FUNCTION_BLOCK _REAL_TestSuite EXTENDS TcUnit.FB_TestSuite
VAR
END_VAR

TestAddress();
TestClearReference();
TestClone();
TestTypeNameReturnsExpected();
TestIsFloat();
TestIsSigned();
TestMakeReferenceToFollowsReference();
TestMakeReferenceToUpdatesReference();
TestSize();
TestValueReturnsExpectedAfterInit();
TestValueReturnsExpectedAfterChange();
TestSerializeTypeWith();
TestSerializeWith();
TestTryDeserializeFrom();
TestTryMakeReferenceToFollowsReference();
TestTryMakeReferenceToUpdatesReference();

METHOD PUBLIC TestAddress
VAR
    _type : _REAL(0.0);
    notExpected : PVOID := 0;
    actual : PVOID;
END_VAR
TEST('TestAddress');

actual := _type.Address;

AssertFalse(
    Condition := (notExpected = actual),
    Message := 'Type did not return a valid address.'
);

TEST_FINISHED();
END_METHOD

METHOD PUBLIC TestClearReference
VAR
    _type : _REAL(0.0);
	target : REAL := 0.0;
    expected : REAL := 0.0;
    actual : REAL;
END_VAR
TEST('TestClearReference');

_type.MakeReferenceTo(target);
_type.ClearReference();
target := 123.4;

actual := _type.Value;

AssertEquals_REAL(
    Expected := expected,
    Actual := actual,
    Delta := REAL#0.001,
    Message := 'Value incorrectly followed target change'
);

TEST_FINISHED();
END_METHOD

METHOD PUBLIC TestClone
VAR
    _type : _REAL(123.4);
	clone : I_Datatype;
	isValidClone : BOOL;
	compareResult : DINT;
END_VAR
TEST('TestClone');

clone := _type.Clone();

isValidClone := clone <> 0;

IF isValidClone THEN
	compareResult := memcmp(_type.Address, clone.Address, clone.Size);
END_IF

AssertTrue(
	Condition := isValidClone,
	Message := 'Clone did not produce a clone'
);

AssertEquals_DINT(
	Expected := 0,
    Actual := compareResult,
    Message := 'Clone did not return a valid clone.'
);

clone.Dispose();

TEST_FINISHED();
END_METHOD

METHOD PUBLIC TestIsFloat
VAR
    _type : _REAL(0);
END_VAR
TEST('TestIsFloat');

AssertTrue(
	Condition := _type.IsFloat,
    Message := 'Type did not correctly identify itself as being unsigned'
);

TEST_FINISHED();
END_METHOD

METHOD PUBLIC TestIsSigned
VAR
    _type : _REAL(0);
END_VAR
TEST('TestIsSigned');

AssertTrue(
	Condition := _type.IsSigned,
    Message := 'Type did not correctly identify itself as being signed'
);

TEST_FINISHED();
END_METHOD

METHOD PUBLIC TestMakeReferenceToFollowsReference
VAR
    _type : _REAL(0.0);
	target : REAL := 0.0;
    expected : REAL := 123.4;
    actual : REAL;
END_VAR
TEST('TestMakeReferenceToFollowsReference');

_type.MakeReferenceTo(target);
target := 123.4;

actual := _type.Value;

AssertEquals_REAL(
    Expected := expected,
    Actual := actual,
    Delta := REAL#0.001,
    Message := 'Value did not follow target change'
);

TEST_FINISHED();
END_METHOD

METHOD PUBLIC TestMakeReferenceToUpdatesReference
VAR
    _type : _REAL(0.0);
	target : REAL := 0.0;
    expected : REAL := 123.4;
    actual : REAL;
END_VAR
TEST('TestMakeReferenceToUpdatesReference');

_type.MakeReferenceTo(target);
_type.Value := 123.4;

actual := target;

AssertEquals_REAL(
    Expected := expected,
    Actual := actual,
    Delta := REAL#0.001,
    Message := 'Value did not update target'
);

TEST_FINISHED();
END_METHOD

METHOD PUBLIC TestSerializeTypeWith
VAR
    _type : _REAL(0.0);
    serializer : JsonSerializer;
    expected : STRING(500) := '{"typeName":"REAL","minValue":-3.4028230607370967e38,"maxValue":3.4028230607370967e38,"isSigned":true,"isFloat":true}';
    actual : STRING(500);
END_VAR
TEST('TestSerializeTypeWith');

serializer.Reset();
_type.SerializeTypeWith(serializer);
serializer.TryGetSerializedData(ADR(actual), SIZEOF(actual));

AssertEquals_STRING(
    Expected := expected,
    Actual := actual,
    Message := 'Serialization of type did not return correct string.'
);

TEST_FINISHED();
END_METHOD

METHOD PUBLIC TestSerializeWith
VAR
    _type : _REAL(123.4);
    serializer : JsonSerializer;
    expected : STRING := '123.4000015258789'; // Expected value due to the nature of floating point values defined by IEEE754.
    actual : STRING(500);
END_VAR
TEST('TestSerializeWith');

serializer.Reset();
_type.SerializeWith(serializer);
serializer.TryGetSerializedData(ADR(actual), SIZEOF(actual));

AssertEquals_STRING(
    Expected := expected,
    Actual := actual,
    Message := 'Serialization of type data did not return correct string.'
);

TEST_FINISHED();
END_METHOD

METHOD PUBLIC TestSize
VAR
    _type : _REAL(0.0);
    expected : UDINT := SIZEOF(REAL);
    actual : UDINT;
END_VAR
TEST('TestSize');

actual := _type.Size;

AssertEquals_UDINT(
    Expected := Expected,
    Actual := actual,
    Message := 'Type did not return the correct size.'
);

TEST_FINISHED();
END_METHOD

METHOD PUBLIC TestTryDeserializeFrom
VAR
    deserializer : JsonDeserializer;
    feedback : DeserializerFeedback;
    json : STRING := '123.4';
    _type : _REAL(0.0);
    expected : REAL := 123.4;
    actual : REAL;
 END_VAR
TEST('TestTryDeserializeFrom');

deserializer.Reset();
deserializer.TryLoad(json);
_type.TryDeserializeFrom(Deserializer, Feedback);

actual := _type.Value;

AssertEquals_REAL(
    Expected := expected,
    Actual := actual,
    Delta := REAL#0.001,
    Message := 'Type did not deserialize correctly.'
);

TEST_FINISHED();
END_METHOD

METHOD PUBLIC TestTryMakeReferenceToFollowsReference
VAR
    _type : _REAL(0.0);
	target : _REAL(0.0);
    expected : REAL := 123.4;
    actual : REAL;
END_VAR
TEST('TestTryMakeReferenceToFollowsReference');

_type.TryMakeReferenceTo(target);
target.Value := 123.4;

actual := _type.Value;

AssertEquals_REAL(
    Expected := expected,
    Actual := actual,
    Delta := REAL#0.001,
    Message := 'Value did not follow target change'
);

TEST_FINISHED();
END_METHOD

METHOD PUBLIC TestTryMakeReferenceToUpdatesReference
VAR
    _type : _REAL(0.0);
	target : _REAL(0.0);
    expected : REAL := 123.4;
    actual : REAL;
END_VAR
TEST('TestTryMakeReferenceToUpdatesReference');

_type.TryMakeReferenceTo(target);
_type.Value := 123.4;

actual := target.Value;

AssertEquals_REAL(
    Expected := expected,
    Actual := actual,
    Delta := REAL#0.001,
    Message := 'Value did not update target'
);

TEST_FINISHED();
END_METHOD

METHOD PUBLIC TestTypeNameReturnsExpected
VAR
    _type : _REAL(0.0);
    expected : STRING := 'REAL';
    actual : STRING;
END_VAR
TEST('TestTypeNameReturnsExpected');

actual := _type.TypeName;

AssertEquals_STRING(
    Expected := expected,
    Actual := actual,
    Message := 'Type did not return correct iec type.'
);

TEST_FINISHED();
END_METHOD

METHOD PUBLIC TestValueReturnsExpectedAfterChange
VAR
    _type : _REAL(0.0);
    expected : REAL := 123.4;
    actual : REAL;
END_VAR
TEST('TestValueReturnsExpectedAfterChange');

_type.Value := 123.4;

actual := _type.Value;

AssertEquals_REAL(
    Expected := expected,
    Actual := actual,
    Delta := REAL#0.001,
    Message := 'Expected value not returned after change.'
);

TEST_FINISHED();
END_METHOD

METHOD PUBLIC TestValueReturnsExpectedAfterInit
VAR
    _type : _REAL(123.4);
    expected : REAL := 123.4;
    actual : REAL;
END_VAR
TEST('TestValueReturnsExpectedAfterInit');

actual := _type.Value;

AssertEquals_REAL(
    Expected := expected,
    Actual := actual,
    Delta := REAL#0.001,
    Message := 'Expected value not returned after Init.'
);

TEST_FINISHED();
END_METHOD

END_FUNCTION_BLOCK

(* stored: Version 1.1.0.1, ProductVersion 3.1.4024.12
   POU _REAL_TestSuite: Id {328b2bf2-c951-05ec-1c81-0c69e5069561}, SpecialFunc None
   Method TestAddress: Id {610e7c27-8321-0728-2089-a702be071d05}
   Method TestClearReference: Id {fed68d47-4e63-0fad-14b3-62b5a8952dbf}
   Method TestClone: Id {0127e830-3223-0ae5-26cb-b68f8efbc94c}
   Method TestIsFloat: Id {55b7a347-680a-4282-9f0e-b6faf433ba3d}
   Method TestIsSigned: Id {6fed8012-e50c-03b8-18f2-dbcc28fe1cd9}
   Method TestMakeReferenceToFollowsReference: Id {bcae6ed8-52cc-06aa-22c8-019b3516c8f2}
   Method TestMakeReferenceToUpdatesReference: Id {0db9ce7e-4897-0740-021e-8239fda97f46}
   Method TestSerializeTypeWith: Id {81939243-ea80-0f98-0994-39b59a5227ca}
   Method TestSerializeWith: Id {fb9dd60e-0eca-072f-2475-b45cd2c0179f}
   Method TestSize: Id {de3ed70c-eb06-03c8-236c-c16748e525fd}
   Method TestTryDeserializeFrom: Id {01f4f376-c22f-0ce1-19b5-32495cdc9da3}
   Method TestTryMakeReferenceToFollowsReference: Id {cfe36170-9938-0837-2a87-419a18b32ca3}
   Method TestTryMakeReferenceToUpdatesReference: Id {a7f19ee6-9b7c-0f36-0d04-dffc930b79aa}
   Method TestTypeNameReturnsExpected: Id {ebaecb80-18bd-0fc1-1124-d7ffd7983c9c}
   Method TestValueReturnsExpectedAfterChange: Id {273c7472-1b95-0705-1f9a-7806c7819252}
   Method TestValueReturnsExpectedAfterInit: Id {46c01183-485e-0cb8-232a-7a0fb5c21738} *)
